// TwinCAT 3 PLC project HMI_PLC
// ProgramVersion: 3.1.4024.0
// CompilerDefines: VISU_USEWSTRING
// libraries:
//   Tc2_Standard, * (Beckhoff Automation GmbH)
//   Tc2_System, * (Beckhoff Automation GmbH)
//   Tc3_JsonXml, * (Beckhoff Automation GmbH)
//   Tc3_Module, * (Beckhoff Automation GmbH)
//   VisuDialogs, * (System)
//   VisuSymbols,3.5.10.0,System
// project tree:
//   Gantry/DUTs/ E_Gantry_State.TcDUT, E_Servo_State.TcDUT, ST_Gantry_Status.TcDUT, ST_Move_Description.TcDUT, ST_Position.TcDUT, ST_Servo_Status.TcDUT
//   Gantry/ FB_Gantry.TcPOU, FB_Servo.TcPOU
//   / GlobalTextList.TcGTLO, GVL.TcGVL, PlcTask.TcTTO (not stored), VISU_TASK.TcTTO
//   POUs/DUTs/ fromHMI.TcDUT, Station_State.TcDUT, toHMI.TcDUT
//   POUs/ HMI.TcVIS, MAIN.TcPOU, VisualizationManager.TcVMO (not stored)
// real-time tasks:
//   TASK PlcTask: cycle T#10ms, priority 20, ADS port 350
//   TASK VISU_TASK: cycle T#200000us, priority 30, ADS port 351

CONFIGURATION HMI_PLC
    RESOURCE PLC ON TwinCAT3
        TASK VISU_TASK(INTERVAL := T#200000us, PRIORITY := 30);
        PROGRAM VisuElems_Visu_Prg WITH VISU_TASK : VisuElems.Visu_Prg;
    END_RESOURCE
END_CONFIGURATION

// ---- Gantry/DUTs/E_Gantry_State.TcDUT
TYPE E_Gantry_State :
(
    DISABLED := 0,      // all motors off
    ENABLING := 10,     // powering up
    HOME_NEEDED := 15,  // on but position unknown
    HOMING := 20,       // finding home
    READY := 30,        // ready for commands
    MOVING := 40,       // moving to target
    STOPPING := 45,     // slowing down
    ERRORED := 100,     // something wrong
    RESETTING := 110    // clearing errors
);
END_TYPE

// ---- Gantry/DUTs/E_Servo_State.TcDUT
TYPE E_Servo_State :
(
    DISABLED := 0,      // motor off
    ENABLING := 10,     // turning on
    HOME_NEEDED := 15,  // on but position unknown
    HOMING := 20,       // finding home
    READY := 30,        // ready for commands
    MOVING := 40,       // moving to target
    STOPPING := 45,     // slowing down
    ERRORED := 100,     // something wrong
    RESETTING := 110    // clearing errors
);
END_TYPE

// ---- Gantry/DUTs/ST_Gantry_Status.TcDUT
{attribute 'OPC.UA.DA' := '1'}
TYPE ST_Gantry_Status :
STRUCT
	// State
	state: E_Gantry_State; // current state
	state_text: STRING; // text display of state
	
	// status flags, only what state doesnt tell us
	all_homed: BOOL; // all axes found home
	at_position: BOOL; // within tolerance of target
	has_error: BOOL; // true if any servo is in error state
	
	// Current position
	position: ST_Position; // where gantry is now
END_STRUCT
END_TYPE

// ---- Gantry/DUTs/ST_Move_Description.TcDUT
{attribute 'OPC.UA.DA' := '1'}
TYPE ST_Move_Description :
STRUCT
	accel: LREAL; 
	decel: LREAL; 
	speed: LREAL; 
	max_torque: LREAL; 
END_STRUCT
END_TYPE

// ---- Gantry/DUTs/ST_Position.TcDUT
{attribute 'OPC.UA.DA' := '1'}
TYPE ST_Position :
STRUCT
	x: LREAL; 
	y: LREAL; 
	z: LREAL; 
END_STRUCT
END_TYPE

// ---- Gantry/DUTs/ST_Servo_Status.TcDUT
TYPE ST_Servo_Status :
STRUCT
	// These can be determined from state
	error_id: DINT; // error code if error is present
	
	// Status flags that state doesn't indicate
	homed: BOOL; // servo is homed/referenced
	at_position: BOOL; // at target position 
	at_home_position: BOOL; // at home position
	
	// Physical values
	actual_position: LREAL; // current position
	actual_velocity: LREAL; // current velocity
	actual_torque: LREAL; // current torque
	
	// Display text
	state_text: STRING; // text for hmi
END_STRUCT
END_TYPE

// ---- POUs/DUTs/fromHMI.TcDUT
TYPE fromHMI :
STRUCT
	cmdReset		: BOOL;		// reset the system
	cmdHome			: BOOL;		// home the system
	cmdAbort		: BOOL;		// abort the system
	cmdStart		: BOOL;		// start the system
	stsReboot		: BOOL;		// HMI rebooting
	stsPointSelected	: ARRAY[0..1] OF INT;	// point selected on the HMI (x,y)
END_STRUCT
END_TYPE

// ---- POUs/DUTs/Station_State.TcDUT
{attribute 'qualified_only'}
{attribute 'strict'}
TYPE Station_State :
(
	RUNNING := 0,
	STOPPED := 1,
	IDLE := 2,
	FAULTED := 3,
	HOMING := 4,
	RESETTING := 5
);
END_TYPE

// ---- POUs/DUTs/toHMI.TcDUT
TYPE toHMI :
STRUCT
	stsController		: INT;	// running, stopped, paused and faulted
	stsPartSelected		: INT;	// part number selected
	stsState		: INT;	// state/step of program
END_STRUCT
END_TYPE

// ---- GVL.TcGVL
VAR_GLOBAL
	// parts coordinates [part_index, coordinate_index]
	// coordinate_index: 1=X_min, 2=Y_min, 3=X_max, 4=Y_max
	Parts : ARRAY[1..4, 1..4] OF INT := [
		30,  700, 180, 850,  // Part 1
		650, 750, 750, 870,  // Part 2 
		50,  20,  250, 120,  // Part 3
		500, 500, 700, 550   // Part 4
	];	
END_VAR

// ---- Gantry/FB_Gantry.TcPOU
{attribute 'hide_all_locals'}
(* 
simple implementation of a 2 axis gantry 
simulating most things for now, pending to do mapping to real servo drive tags,
do specific behaivor handling based on servo model and error handling
*)

FUNCTION_BLOCK FB_Gantry
VAR_IN_OUT
	// control inputs

	pcmd_enable: BOOL; // power up all axes
	pcmd_disable: BOOL; // shut down all axes
	pcmd_home: BOOL; // find home for all axes
	pcmd_reset_error: BOOL; // clear errors
	pcmd_move_absolute: BOOL; // go to exact position
	pcmd_stop: BOOL; // stop moving
END_VAR
VAR_INPUT	
	// setup options
	cfg_simulation_mode: BOOL := TRUE; // just simulate no hardware
	cfg_position_tolerance: LREAL := 0.05; // how close is close enough mm
	
	// gantry limits and home position
	cfg_max_x: LREAL := 1000.0; // max x position in mm
	cfg_max_y: LREAL := 1000.0; // max y position in mm
	cfg_home_offset_x: LREAL := 10.0; // home position x offset in mm
	cfg_home_offset_y: LREAL := 10.0; // home position y offset in mm
	
	// movement targets
	inp_target_position: ST_Position; // where to go
	inp_move_description: ST_Move_Description; // how fast to go
END_VAR

VAR_OUTPUT
	// status info
	sts: ST_Gantry_Status; // everything about current state
END_VAR

VAR
	// motion profiles for each axis
	internal_move_desc_x: ST_Move_Description;
	internal_move_desc_y: ST_Move_Description;
	
	// the actual motors
	x_axis: FB_Servo;
	y_axis: FB_Servo;
	
	// x-axis controls
	cmd_x_enable: BOOL;
	cmd_x_disable: BOOL;
	cmd_x_home: BOOL;
	cmd_x_reset_error: BOOL;
	cmd_x_move_absolute: BOOL;
	cmd_x_stop: BOOL;
	
	// y-axis controls
	cmd_y_enable: BOOL;
	cmd_y_disable: BOOL;
	cmd_y_home: BOOL;
	cmd_y_reset_error: BOOL;
	cmd_y_move_absolute: BOOL;
	cmd_y_stop: BOOL;
END_VAR

// update status first to get current axis states
Update_Status();

// use same speed settings for all axes
internal_move_desc_x := inp_move_description;
internal_move_desc_y := inp_move_description;

// check errors first using the has_error flag
IF sts.has_error AND NOT pcmd_reset_error THEN
    // stuck in error until reset
    sts.state := E_Gantry_State.ERRORED;
    
// nothing else happens while in error
ELSE
    // main state machine
    CASE sts.state OF
        E_Gantry_State.DISABLED:
            // when disabled we can only enable
            IF pcmd_enable AND NOT sts.has_error THEN
                sts.state := E_Gantry_State.ENABLING;
            END_IF
            
        E_Gantry_State.ENABLING:
            // turn on all motors
            cmd_x_enable := TRUE;
            cmd_y_enable := TRUE;
            
            // once all are not disabled we need to find home
            IF x_axis.sts_State <> E_Servo_State.DISABLED AND 
               y_axis.sts_State <> E_Servo_State.DISABLED THEN
                sts.state := E_Gantry_State.HOME_NEEDED;
            END_IF
            
        E_Gantry_State.HOME_NEEDED:
            // start homing when requested
            IF pcmd_home THEN
                sts.state := E_Gantry_State.HOMING;
                
                // tell all axes to find home
                cmd_x_home := TRUE;
                cmd_y_home := TRUE;
            ELSIF pcmd_disable THEN
                sts.state := E_Gantry_State.DISABLED;
                
                // turn everything off
                cmd_x_disable := TRUE;
                cmd_y_disable := TRUE;
            END_IF
            
        E_Gantry_State.HOMING:
            // handle stop during homing
            IF pcmd_stop THEN
                sts.state := E_Gantry_State.HOME_NEEDED;
                
                // tell all axes to halt
                cmd_x_stop := TRUE;
                cmd_y_stop := TRUE;
            
            // when all axes found home good to go
            ELSIF sts.all_homed AND 
                  x_axis.sts_State <> E_Servo_State.MOVING AND 
                  y_axis.sts_State <> E_Servo_State.MOVING THEN
                
                // move to home offset position if homed
                sts.state := E_Gantry_State.MOVING;
                
                // set target to home offset
                inp_target_position.x := cfg_home_offset_x;
                inp_target_position.y := cfg_home_offset_y;
                
                // move to home offset
                cmd_x_move_absolute := TRUE;
                cmd_y_move_absolute := TRUE;
            END_IF
            
        E_Gantry_State.READY:
            // handle shutdown request
            IF pcmd_disable THEN
                sts.state := E_Gantry_State.DISABLED;
                
                // turn everything off
                cmd_x_disable := TRUE;
                cmd_y_disable := TRUE;
            
            // rehome if needed
            ELSIF pcmd_home THEN
                sts.state := E_Gantry_State.HOMING;
                
                // tell all axes to find home
                cmd_x_home := TRUE;
                cmd_y_home := TRUE;
                
            // go to exact position
            ELSIF pcmd_move_absolute AND sts.all_homed THEN
                // check if position is within limits
                IF inp_target_position.x > cfg_max_x OR inp_target_position.x < 0 OR
                   inp_target_position.y > cfg_max_y OR inp_target_position.y < 0 THEN
                    // position out of bounds - do not move
                    // could set an error flag here
                ELSE
                    // check if already there
                    sts.at_position := 
                        x_axis.sts.at_position AND 
                        y_axis.sts.at_position;
                    
                    IF sts.at_position THEN
                        // already there nothing to do
                        sts.at_position := TRUE;
                    ELSE
                        sts.state := E_Gantry_State.MOVING;
                        sts.at_position := FALSE;
                        
                        // tell all axes where to go
                        cmd_x_move_absolute := TRUE;
                        cmd_y_move_absolute := TRUE;
                    END_IF
                END_IF
            END_IF
            
        E_Gantry_State.MOVING:
            // handle stop while moving
            IF pcmd_stop THEN
                sts.state := E_Gantry_State.STOPPING;
                
                // tell all axes to halt
                cmd_x_stop := TRUE;
                cmd_y_stop := TRUE;
            
            // when motion complete back to ready
            ELSIF x_axis.sts_State <> E_Servo_State.MOVING AND 
                  y_axis.sts_State <> E_Servo_State.MOVING THEN
                sts.state := E_Gantry_State.READY;
            END_IF
            
        E_Gantry_State.STOPPING:
            // wait until fully stopped
            IF x_axis.sts_State <> E_Servo_State.MOVING AND 
               y_axis.sts_State <> E_Servo_State.MOVING THEN
                sts.state := E_Gantry_State.READY;
            END_IF
            
        E_Gantry_State.ERRORED:
            // reset errors when commanded
            IF pcmd_reset_error THEN
                sts.state := E_Gantry_State.RESETTING;
                
                // tell all axes to clear errors
                cmd_x_reset_error := TRUE;
                cmd_y_reset_error := TRUE;
            END_IF
            
        E_Gantry_State.RESETTING:
            // when all errors cleared go to disabled state
            IF NOT sts.has_error THEN
                sts.state := E_Gantry_State.DISABLED;
            END_IF
    END_CASE;
END_IF;

// now actually run each motor
// x-axis
x_axis(
    // commands
    pcmd_enable := cmd_x_enable,
    pcmd_disable := cmd_x_disable,
    pcmd_home := cmd_x_home,
    pcmd_reset_error := cmd_x_reset_error,
    pcmd_move_absolute := cmd_x_move_absolute,
    pcmd_stop := cmd_x_stop,
	
	// configuration
	cfg_simulation_mode := cfg_simulation_mode,
	cfg_position_tolerance := cfg_position_tolerance,
	
	// movement parameters
	inp_target_position := inp_target_position.x,
	inp_move_description := internal_move_desc_x
);

// y-axis
y_axis(
    // commands
    pcmd_enable := cmd_y_enable,
    pcmd_disable := cmd_y_disable,
    pcmd_home := cmd_y_home,
    pcmd_reset_error := cmd_y_reset_error,
    pcmd_move_absolute := cmd_y_move_absolute,
    pcmd_stop := cmd_y_stop,
	
	// configuration
	cfg_simulation_mode := cfg_simulation_mode,
	cfg_position_tolerance := cfg_position_tolerance,
	
	// movement parameters
	inp_target_position := inp_target_position.y,
	inp_move_description := internal_move_desc_y
);

// update status again after running motors
Update_Status();

Reset_Commands();

METHOD Reset_Commands : BOOL
VAR_INPUT
END_VAR
// reset button presses one pulse per press
IF pcmd_enable THEN pcmd_enable := FALSE; END_IF;
IF pcmd_disable THEN pcmd_disable := FALSE; END_IF;
IF pcmd_home THEN pcmd_home := FALSE; END_IF;
IF pcmd_reset_error THEN pcmd_reset_error := FALSE; END_IF;
IF pcmd_move_absolute THEN pcmd_move_absolute := FALSE; END_IF;
IF pcmd_stop THEN pcmd_stop := FALSE; END_IF;
END_METHOD

METHOD Update_Status : BOOL
VAR_INPUT
END_VAR
// update our current position
sts.position.x := x_axis.sts.actual_position;
sts.position.y := y_axis.sts.actual_position;
sts.position.z := 0; // Z axis removed

// update status (only what we can't determine from state)
sts.all_homed := x_axis.sts.homed AND y_axis.sts.homed;

// check if any axis has an error
sts.has_error := x_axis.sts_State = E_Servo_State.ERRORED OR 
                y_axis.sts_State = E_Servo_State.ERRORED;

// set target position status - are we there yet?
IF sts.state = E_Gantry_State.READY THEN
    sts.at_position := 
        x_axis.sts.at_position AND 
        y_axis.sts.at_position;
ELSIF sts.state <> E_Gantry_State.MOVING THEN
    // when not moving or ready not at any target
    sts.at_position := FALSE;
END_IF;

// set state text for hmi display
CASE sts.state OF
    E_Gantry_State.DISABLED:
        sts.state_text := 'DISABLED';
    E_Gantry_State.ENABLING:
        sts.state_text := 'ENABLING';
    E_Gantry_State.HOME_NEEDED:
        sts.state_text := 'HOME NEEDED';
    E_Gantry_State.HOMING:
        sts.state_text := 'HOMING';
    E_Gantry_State.READY:
        sts.state_text := 'READY';
    E_Gantry_State.MOVING:
        sts.state_text := 'MOVING';
    E_Gantry_State.STOPPING:
        sts.state_text := 'STOPPING';
    E_Gantry_State.ERRORED:
        sts.state_text := 'ERROR';
    E_Gantry_State.RESETTING:
        sts.state_text := 'RESETTING';
ELSE
    sts.state_text := 'UNKNOWN';
END_CASE;
END_METHOD

END_FUNCTION_BLOCK

// ---- Gantry/FB_Servo.TcPOU
{attribute 'hide_all_locals'}
FUNCTION_BLOCK FB_Servo
VAR_IN_OUT
	// button inputs
	pcmd_enable: BOOL; // turn on motor
	pcmd_disable: BOOL; // turn off motor
	pcmd_home: BOOL; // find home position
	pcmd_reset_error: BOOL; // clear errors
	pcmd_move_absolute: BOOL; // go to exact position
	pcmd_stop: BOOL; // stop moving
END_VAR

VAR_INPUT
	// setup options
	cfg_simulation_mode: BOOL := TRUE; // just simulate no hardware
	cfg_home_position: LREAL := 0; // where home is
	cfg_position_tolerance: LREAL := 0.05; // how close is close enough
	
	// movement inputs
	inp_target_position: LREAL; // where to go
	inp_Move_Description: ST_Move_Description; // how fast to get there
END_VAR

VAR_OUTPUT
	// info for hmi and other functions
	sts: ST_Servo_Status; // full status structure
	sts_State: E_Servo_State; // current state
	
	// movement type flags
	sts_absolute_move: BOOL; // going to exact position
END_VAR

VAR
	// working variables
	internal_target_position: LREAL; // where we headed
	internal_sim_timer: TON; // for simulating movements
	internal_sim_home_timer: TON; // for simulating homing
	internal_sim_reset_timer: TON; // for simulating reset
	internal_sim_stop_timer: TON; // for simulating stopping
	internal_sim_move_time: TIME; // how long move takes
	internal_error_timer: TON; // for simulating random errors
	
	// motion calculation vars
	internal_start_position: LREAL; // where we started
	internal_position_delta: LREAL; // how far to move
	
	// helpers
	temp_ratio: LREAL; // for position interpolation
END_VAR

// errors trump everything else
IF sts_State = E_Servo_State.ERRORED AND NOT pcmd_reset_error AND sts_State <> E_Servo_State.RESETTING THEN
    // stuck in error until reset
    sts_State := E_Servo_State.ERRORED;
    
    // nothing happens while in error
ELSE
    // main state machine
    CASE sts_State OF
        E_Servo_State.DISABLED: // power off
            IF pcmd_enable AND sts_State <> E_Servo_State.ERRORED THEN
                sts_State := E_Servo_State.ENABLING; // power up
            END_IF
            
        E_Servo_State.ENABLING: // powering up
            IF cfg_simulation_mode THEN
                // pretend to power up
                // dont know where we are yet
                sts_State := E_Servo_State.HOME_NEEDED;
            ELSE
                // TODO: actually turn on real servo
            END_IF
            
        E_Servo_State.HOME_NEEDED: // need to find home
            // can either go home or shut down
            IF pcmd_disable THEN
                sts_State := E_Servo_State.DISABLED;
            ELSIF pcmd_home THEN
                sts_State := E_Servo_State.HOMING;
                sts.homed := FALSE;
                
                IF cfg_simulation_mode THEN
                    // pretend to home for 2 seconds
                    internal_sim_home_timer(IN := FALSE); // reset timer
                    internal_sim_home_timer(IN := TRUE, PT := T#2S); // start timer with 2s delay
                END_IF
            END_IF
            
        E_Servo_State.HOMING: // looking for home
            IF pcmd_stop THEN
                // cancelled homing
                sts_State := E_Servo_State.HOME_NEEDED; // back to square one
                RETURN;
            END_IF
            
            IF cfg_simulation_mode THEN
                // pretend to find home
                internal_sim_home_timer();
                
                IF internal_sim_home_timer.Q THEN
                    // found home
                    sts.homed := TRUE;
                    sts.actual_position := cfg_home_position;
                    sts.at_home_position := TRUE;
                    sts_State := E_Servo_State.READY; // good to go
                END_IF
            ELSE
                // TODO: actually find home with real hardware
            END_IF
            
        E_Servo_State.READY: // ready for action
            IF pcmd_disable THEN
                // shut it down
                sts_State := E_Servo_State.DISABLED;
            ELSIF pcmd_home THEN
                // find home again
                sts_State := E_Servo_State.HOMING;
                sts.homed := FALSE;
                
                IF cfg_simulation_mode THEN
                    // pretend to home again for 2 seconds
                    internal_sim_home_timer(IN := FALSE); // reset timer
                    internal_sim_home_timer(IN := TRUE, PT := T#2S); // start timer with 2s delay
                END_IF
            ELSIF pcmd_move_absolute THEN
                // check if already there
                IF ABS(inp_target_position - sts.actual_position) <= cfg_position_tolerance THEN
                    // already here no need to move
                    sts.at_position := TRUE;
                ELSE
                    // go to exact position
                    internal_target_position := inp_target_position;
                    internal_start_position := sts.actual_position;
                    internal_position_delta := internal_target_position - internal_start_position;
                    sts_State := E_Servo_State.MOVING;
                    sts.at_position := FALSE;
                    
                    // set move type
                    sts_absolute_move := TRUE;
                    
                    IF cfg_simulation_mode THEN
                        // figure out how long move should take
                        internal_sim_move_time := LREAL_TO_TIME(ABS(internal_position_delta) / 
                                                              (inp_Move_Description.speed) * 1000);
                        // make sure not too quick
                        IF internal_sim_move_time < T#100MS THEN
                            internal_sim_move_time := T#100MS;
                        END_IF
                        
                        // set up move timer
                        internal_sim_timer(IN := FALSE); // reset timer
                        internal_sim_timer(IN := TRUE, PT := internal_sim_move_time); // start timer
                    END_IF
                END_IF
            END_IF
            
        E_Servo_State.MOVING: // moving to target
            // handle stop command
            IF pcmd_stop THEN
                sts_State := E_Servo_State.STOPPING;
                // Keep position where it is - no need for timer
                sts.actual_velocity := 0;
                RETURN;
            END_IF
            
            IF cfg_simulation_mode THEN
                // fake the movement
                internal_sim_timer();
                
                // calculate position during move
                IF NOT internal_sim_timer.Q THEN
                    // how far along are we
                    // TIME_TO_REAL gives milliseconds
                    temp_ratio := TIME_TO_REAL(internal_sim_timer.ET) / TIME_TO_REAL(internal_sim_move_time);
                    
                    // cap at 100%
                    IF temp_ratio > 1.0 THEN 
                        temp_ratio := 1.0;
                    END_IF;
                    
                    // linear position: start + (distance * percentage)
                    sts.actual_position := internal_start_position + (internal_position_delta * temp_ratio);
                    sts.actual_velocity := inp_Move_Description.speed;
                    sts.actual_torque := inp_Move_Description.max_torque * 0.5; // about half torque
                ELSE
                    // made it
                    sts.actual_position := internal_target_position;
                    sts.actual_velocity := 0;
                    sts.actual_torque := 0;
                    sts.at_position := TRUE;
                    sts_State := E_Servo_State.READY; // back to ready
                END_IF
            ELSE
                // TODO: move real motor to position
            END_IF
            
        E_Servo_State.STOPPING: // stopping movement
            // Immediately stop movement and transition to READY
            sts.actual_velocity := 0;
            sts_State := E_Servo_State.READY;
            
        E_Servo_State.ERRORED: // error condition
            // reset button pressed
            IF pcmd_reset_error THEN
                sts_State := E_Servo_State.RESETTING;
                
                // set up reset timer
                IF cfg_simulation_mode THEN
                    internal_sim_reset_timer(IN := FALSE); // reset timer
                    internal_sim_reset_timer(IN := TRUE, PT := T#1S); // start timer with 1s delay
                END_IF
            END_IF
            
        E_Servo_State.RESETTING: // clearing errors
            // wait for reset to complete
            IF cfg_simulation_mode THEN
                internal_sim_reset_timer();
                
                IF internal_sim_reset_timer.Q THEN
                    // all better now
                    sts_State := E_Servo_State.DISABLED;
                END_IF
            ELSE
                // TODO: actually reset hardware
            END_IF
    END_CASE
END_IF;

// set state text for hmi display
CASE sts_State OF
    E_Servo_State.DISABLED:
        sts.state_text := 'DISABLED';
    E_Servo_State.ENABLING:
        sts.state_text := 'ENABLING';
    E_Servo_State.HOME_NEEDED:
        sts.state_text := 'HOME NEEDED';
    E_Servo_State.HOMING:
        sts.state_text := 'HOMING';
    E_Servo_State.READY:
        sts.state_text := 'READY';
    E_Servo_State.MOVING:
        IF sts_absolute_move THEN
            sts.state_text := 'MOVING TO POSITION';
        ELSE
            sts.state_text := 'MOVING';
        END_IF
    E_Servo_State.STOPPING:
        sts.state_text := 'STOPPING';
    E_Servo_State.ERRORED:
        sts.state_text := 'ERROR';
    E_Servo_State.RESETTING:
        sts.state_text := 'RESETTING';
ELSE
    sts.state_text := 'UNKNOWN';
END_CASE;

// check if at home
sts.at_home_position := (ABS(sts.actual_position - cfg_home_position) < 0.001);

// check if at target
sts.at_position := (ABS(sts.actual_position - inp_target_position) <= cfg_position_tolerance);

// reset button flags one press per command
IF pcmd_enable THEN pcmd_enable := FALSE; END_IF;
IF pcmd_disable THEN pcmd_disable := FALSE; END_IF;
IF pcmd_home THEN pcmd_home := FALSE; END_IF;
IF pcmd_reset_error THEN pcmd_reset_error := FALSE; END_IF;
IF pcmd_move_absolute THEN pcmd_move_absolute := FALSE; END_IF;
IF pcmd_stop THEN pcmd_stop := FALSE; END_IF;

METHOD SimulateRandomErrors
VAR_INPUT
END_VAR
(*
we could get the error list form the drive manual and have an enum here to simulate different types
of errors, show on the HMI and do error handling ahead of comissioning 

*)


// only in simulation mode and not in error state
IF cfg_simulation_mode AND sts_State <> E_Servo_State.ERRORED THEN
    // set up error timer random interval
    internal_error_timer(IN := TRUE, PT := T#30S);
    
    // generate error after timer expires
    IF internal_error_timer.Q THEN
        sts.error_id := 1000; // generic error code
        sts_State := E_Servo_State.ERRORED; // go to error state
        
        // reset timer
        internal_error_timer(IN := FALSE);
    END_IF
END_IF
END_METHOD

END_FUNCTION_BLOCK

// ---- POUs/MAIN.TcPOU
PROGRAM MAIN
VAR
	// Our gantry controller
	my_gantry: FB_Gantry;
	
	
	// Where to move to
	target_position: ST_Position;
	
	// Speed settings
	move_params: ST_Move_Description := (speed:= 5 , accel := 10, decel := 10, max_torque := 80);
	
	// HMI Tags
	api_fromHMI : fromHMI;
	api_toHMI : toHMI;

	// Internal tags for gantry control
	cmd_enable: BOOL;
	cmd_disable: BOOL;
	cmd_home: BOOL;
	cmd_move_to_position: BOOL;
	cmd_stop: BOOL;
	cmd_reset_error: BOOL;
	
	// actuator command for pen ( TODO implement actuator FB )
	cmd_penAdvance : BOOL := FALSE;
	
	// Process state machine
	process_state : INT := 0;
	selected_part : INT := 0;
	drawing_complete : BOOL := FALSE;

	
	// Draw_Part method variables
	draw_local_corner : INT := 1;
	draw_local_wait_timer : TON;
	draw_local_wait_time : TIME := T#500MS;
	draw_local_state : INT := 0;
	draw_local_done : BOOL := FALSE;
END_VAR

// Update HMI at the top
Update_HMI();

my_gantry(
    pcmd_enable := cmd_enable,
    pcmd_disable := cmd_disable,
    pcmd_home := cmd_home,
    pcmd_move_absolute := cmd_move_to_position,
    pcmd_stop := cmd_stop,
    pcmd_reset_error := cmd_reset_error,

    cfg_simulation_mode := TRUE,
    inp_target_position := target_position,
    inp_move_description := move_params
);

// Check if point from HMI is inside any part
api_toHMI.stsPartSelected := Find_Part(
        x := DINT_TO_LREAL(api_fromHMI.stsPointSelected[0]),
        y := DINT_TO_LREAL(api_fromHMI.stsPointSelected[1]));

// Main process state machine
CASE process_state OF
    0: // just starting up
        // jump to idle
        process_state := 10;
        api_toHMI.stsState := 0;
        
    10: // chilling in idle
        // grab selected part
        selected_part := api_toHMI.stsPartSelected;
        api_toHMI.stsState := 10;
        
        // handle start button
        IF api_fromHMI.cmdStart AND selected_part > 0 THEN
            // ready to rock if gantry is up
            IF my_gantry.sts.state = E_Gantry_State.READY THEN
                process_state := 20; // go draw
                draw_local_state := 0; // reset drawer
                draw_local_done := FALSE; // not done yet
            ELSIF my_gantry.sts.state = E_Gantry_State.DISABLED THEN
                // wake up gantry first
                cmd_enable := TRUE;
                process_state := 15; // power up sequence
            END_IF;
        END_IF;
        
    15: // getting gantry ready
        api_toHMI.stsState := 15;
        IF my_gantry.sts.state = E_Gantry_State.HOME_NEEDED THEN
            cmd_home := TRUE;
        ELSIF my_gantry.sts.state = E_Gantry_State.READY THEN
            process_state := 10; // back to chilling
        END_IF;
        
    16: // home sequence
        api_toHMI.stsState := 16;
        IF my_gantry.sts.state = E_Gantry_State.DISABLED THEN
            cmd_enable := TRUE;
        ELSIF my_gantry.sts.state = E_Gantry_State.HOME_NEEDED THEN
            cmd_home := TRUE;
        ELSIF my_gantry.sts.state = E_Gantry_State.READY THEN
            process_state := 10; // back to idle
        END_IF;
        
    20: // busy drawing
        api_toHMI.stsState := 20;
        drawing_complete := Draw_Part(selected_part);
        
        // finished the masterpiece
        IF drawing_complete THEN
            process_state := 10; // back to idle
        END_IF;
        
    30: // emergency stop
        api_toHMI.stsState := 30;
        // hit the brakes
        cmd_stop := TRUE;
        // lift the pen
        cmd_penAdvance := FALSE;
        
        // back to idle when stopped
        IF my_gantry.sts.state = E_Gantry_State.READY THEN
            process_state := 10; // back to idle
        END_IF;
END_CASE;

// Global command handling (except during abort)
IF process_state <> 30 THEN
    // abort = stop everything
    IF api_fromHMI.cmdAbort THEN
        process_state := 30; // emergency stop
    END_IF;
    
    // home button pressed
    IF api_fromHMI.cmdHome THEN
        // start home sequence
        process_state := 16;
    END_IF;
    
    // reset button clears errors
    IF api_fromHMI.cmdReset THEN
        cmd_reset_error := TRUE;
    END_IF;
END_IF;

METHOD Draw_Part : BOOL
VAR_INPUT
	part_to_draw : INT := 0;
END_VAR
// If part doesn't exist, exit
IF part_to_draw < 1 OR part_to_draw > 4 THEN
    Draw_Part := FALSE;
    RETURN;
END_IF;

// State machine for drawing the part
CASE draw_local_state OF
    0: // Initial state - Lift pen
		draw_local_done := FALSE;
        cmd_penAdvance := FALSE;
        draw_local_state := 10;
        
    10: // Move to first corner (bottom left)
        target_position.x := GVL.Parts[part_to_draw, 1]; // X_min
        target_position.y := GVL.Parts[part_to_draw, 2]; // Y_min
        cmd_move_to_position := TRUE;
        draw_local_state := 20;
        
    20: // Wait for gantry to reach position
        IF my_gantry.sts.at_position THEN
            draw_local_state := 30;
        END_IF;
        
    30: // Lower pen
        cmd_penAdvance := TRUE;
        draw_local_state := 40;
        
    40: // Move to second corner (bottom right)
        target_position.x := GVL.Parts[part_to_draw, 3]; // X_max
        target_position.y := GVL.Parts[part_to_draw, 2]; // Y_min
        cmd_move_to_position := TRUE;
        draw_local_state := 50;
        
    50: // Wait for gantry to reach position
        IF my_gantry.sts.at_position THEN
            draw_local_state := 60;
        END_IF;
        
    60: // Move to third corner (top right)
        target_position.x := GVL.Parts[part_to_draw, 3]; // X_max
        target_position.y := GVL.Parts[part_to_draw, 4]; // Y_max
        cmd_move_to_position := TRUE;
        draw_local_state := 70;
        
    70: // Wait for gantry to reach position
        IF my_gantry.sts.at_position THEN
            draw_local_state := 80;
        END_IF;
        
    80: // Move to fourth corner (top left)
        target_position.x := GVL.Parts[part_to_draw, 1]; // X_min
        target_position.y := GVL.Parts[part_to_draw, 4]; // Y_max
        cmd_move_to_position := TRUE;
        draw_local_state := 90;
        
    90: // Wait for gantry to reach position
        IF my_gantry.sts.at_position THEN
            draw_local_state := 100;
        END_IF;
        
    100: // Move back to first corner (bottom left) to close the rectangle
        target_position.x := GVL.Parts[part_to_draw, 1]; // X_min
        target_position.y := GVL.Parts[part_to_draw, 2]; // Y_min
        cmd_move_to_position := TRUE;
        draw_local_state := 110;
        
    110: // Wait for gantry to reach position
        IF my_gantry.sts.at_position THEN
            draw_local_state := 120;
        END_IF;
        
    120: // Lift pen and finish
        cmd_penAdvance := FALSE;
        draw_local_state := 130;
        
    130: // Drawing complete
        draw_local_done := TRUE;
        Draw_Part := TRUE;  // Return TRUE to indicate success
        draw_local_state := 0;  // Reset for next drawing
END_CASE;
END_METHOD

METHOD Find_Part : INT
VAR_INPUT
	x : LREAL;
	y : LREAL;
END_VAR
VAR
	i : INT;
END_VAR
// Initialize return value to 0 (no part found)
Find_Part := 0;

// Loop through all parts to check if point is inside any of them
FOR i := 1 TO 4 DO
    // Check if point (x,y) is inside the part boundaries:
    // x >= X_min AND x <= X_max AND y >= Y_min AND y <= Y_max
    IF x >= GVL.Parts[i,1] AND x <= GVL.Parts[i,3] AND
       y >= GVL.Parts[i,2] AND y <= GVL.Parts[i,4] THEN
        Find_Part := i;
        RETURN;
    END_IF;
END_FOR;
END_METHOD

METHOD Update_HMI : BOOL
VAR_INPUT
END_VAR
// Handle HMI commands
IF api_fromHMI.cmdHome THEN
    cmd_home := TRUE;
    api_fromHMI.cmdHome := FALSE; // Reset the HMI command
END_IF;

IF api_fromHMI.cmdReset THEN
    cmd_reset_error := TRUE;
    api_fromHMI.cmdReset := FALSE; // Reset the HMI command
END_IF;

IF api_fromHMI.cmdAbort THEN
    cmd_stop := TRUE;
    cmd_disable := TRUE;
    api_fromHMI.cmdAbort := FALSE; // Reset the HMI command
END_IF;

// cmdStart logic pending for future implementation

// Update HMI status using Station_State enumeration
CASE my_gantry.sts.state OF
    E_Gantry_State.ERRORED: 
        api_toHMI.stsController := Station_State.FAULTED;
    E_Gantry_State.DISABLED, E_Gantry_State.STOPPING:
        api_toHMI.stsController := Station_State.STOPPED;
    E_Gantry_State.MOVING:
        api_toHMI.stsController := Station_State.RUNNING;
    E_Gantry_State.HOMING:
        api_toHMI.stsController := Station_State.HOMING;
    E_Gantry_State.ENABLING:
        api_toHMI.stsController := Station_State.RUNNING;
    E_Gantry_State.RESETTING:
        api_toHMI.stsController := Station_State.RESETTING;
    ELSE
        api_toHMI.stsController := Station_State.IDLE;
END_CASE;
END_METHOD

END_PROGRAM

// ---- GlobalTextList.TcGTLO
TEXTLIST GlobalTextList
  593 = '%.0f'
  548 = '%.s'
  547 = '%d'
  451 = '%s'
  205 = 'Abort'
  24 = 'Controller Status'
  858 = 'Current Position'
  337 = 'DISABLE'
  939 = 'Enable'
  533 = 'ENABLE'
  675 = 'Gantry System'
  744 = 'HOME'
  349 = 'Home'
  885 = 'MOVE'
  3 = 'Not Part of API'
  561 = 'Not Part of API, adding for visu'
  430 = 'Part Selected'
  38 = 'Pen Plotter'
  251 = 'Pen Position'
  313 = 'Point Selected'
  418 = 'Reboot'
  464 = 'RESET'
  188 = 'Reset'
  377 = 'Start'
  383 = 'State'
  538 = 'Status'
  55 = 'STOP'
  459 = 'Target Position'
  851 = 'X Current Position'
  119 = 'X Position'
  323 = 'X Target  Position'
  729 = 'Y Current Position'
  614 = 'Y Target  Position'
  213 = 'Z Current Position'
  86 = 'Z CurrentPosition'
  872 = 'Z Target  Position'
END_TEXTLIST

// ---- POUs/HMI.TcVIS
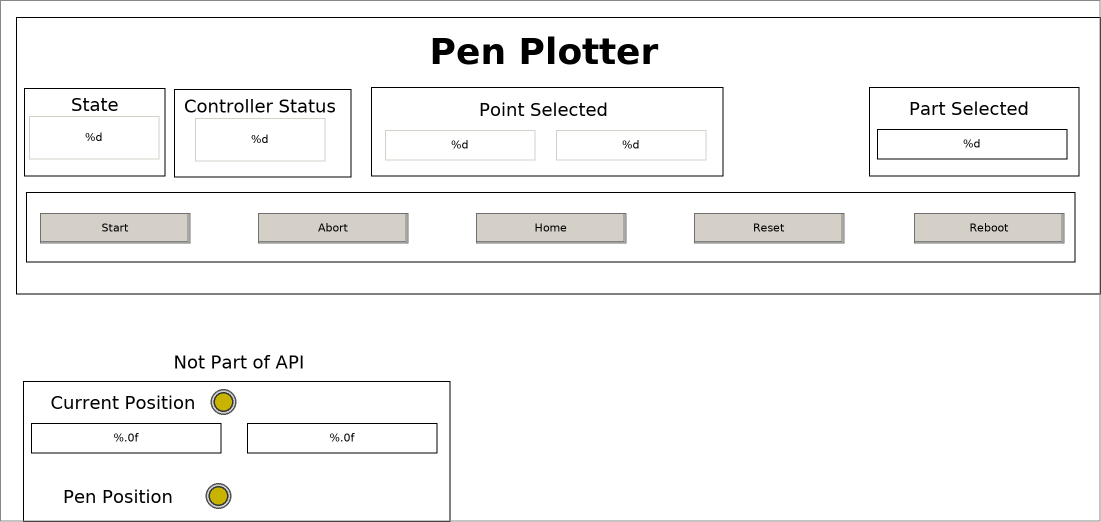
VISUALIZATION HMI  // 1101x522
    RoundedRectangle (16,17 1085x277)
    RoundedRectangle (23,381 427x141)
    Rectangle (247,423 190x30), "%.0f", text variable: MAIN.my_gantry.sts.position.y
    Rectangle (31,423 190x30), "%.0f", text variable: MAIN.my_gantry.sts.position.x
    Lamp1 (205,387 37x30), variable: MAIN.my_gantry.sts.at_position, style: Lamp-Lamp1-Yellow
    Label (28,388 190x30), "Current Position"
    RoundedRectangle (371,87 352x89)
    Textfield (385,130 150x30), "%d", text variable: MAIN.api_fromHMI.stsPointSelected[0]
        OnMouseDown: write the text variable via InputWithLimits, min 0, max 1000, title 'Target Position X'
    Textfield (556,130 150x30), "%d", text variable: MAIN.api_fromHMI.stsPointSelected[1]
        OnMouseDown: write the text variable via InputWithLimits, min 0, max 1000, title 'Target Position X'
    Label (384,95 319x30), "Point Selected"
    RoundedRectangle (24,88 141x88)
    Textfield (29,116 130x43), "%d", text variable: MAIN.api_toHMI.stsState
    Label (28,90 134x30), "State"
    RoundedRectangle (26,192 1049x70)
    Button (914,213 150x30), "Reboot"
        tap MAIN.api_fromHMI.stsReboot
    Button (40,213 150x30), "Start"
        tap MAIN.api_fromHMI.cmdStart p1329445385=TRUE
    Button (258,213 150x30), "Abort"
        tap MAIN.api_fromHMI.cmdAbort p1329445385=TRUE
    Button (476,213 150x30), "Home"
        tap MAIN.api_fromHMI.cmdHome
    Button (694,213 150x30), "Reset"
        tap MAIN.api_fromHMI.cmdReset p1329445385=TRUE
    Label (25,22 1038x59), "Pen Plotter"
    RoundedRectangle (174,89 177x88)
    Textfield (195,118 130x43), "%d", text variable: MAIN.api_toHMI.stsState
    Label (178,93 164x27), "Controller Status"
    Label (26,349 426x27), "Not Part of API"
    RoundedRectangle (869,87 210x89)
    Rectangle (877,129 190x30), "%d", text variable: MAIN.api_toHMI.stsPartSelected
    Label (874,94 190x30), "Part Selected"
    Lamp1 (200,481 37x30), variable: MAIN.cmd_penAdvance, style: Lamp-Lamp1-Yellow
    Label (23,482 190x30), "Pen Position"
END_VISUALIZATION
